FUNCTION_BLOCK CounterSp (* Basic Function Block Type *)
  (* Standard: 61499-2 *)
  (* Version 0.0, 7/15/2026, Schneider Electric, Template *)
  PACKAGE SE.Nereda;
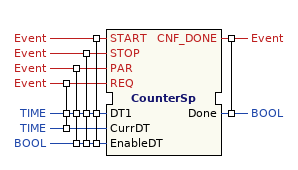
  EVENT_INPUT
    START WITH DT1, EnableDT; (* Normal Execution Request *)
    STOP WITH DT1, EnableDT;
    PAR WITH DT1, EnableDT;
    REQ WITH CurrDT, DT1;
  END_EVENT
  EVENT_OUTPUT
    CNF_DONE WITH Done; (* Execution Confirmation *)
  END_EVENT
  VAR_INPUT
    DT1 : TIME; (* Input event qualifier *)
    CurrDT : TIME;
    EnableDT : BOOL;
  END_VAR
  VAR_OUTPUT
    Done : BOOL; (* Output event qualifier *)
  END_VAR
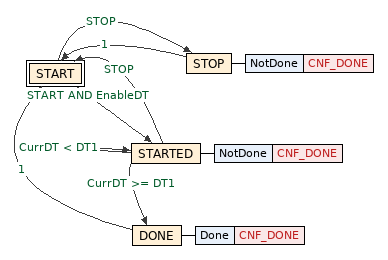
  EC_STATES
    START; (* Initial State *)
    STARTED : NotDone -> CNF_DONE; (* Normal execution *)
    DONE : Done -> CNF_DONE;
    STOP : NotDone -> CNF_DONE;
  END_STATES
  EC_TRANSITIONS
    START TO STARTED := START AND EnableDT;
    STARTED TO STARTED := CurrDT < DT1;
    STARTED TO DONE := CurrDT >= DT1;
    DONE TO START := 1;
    STARTED TO START := STOP;
    START TO STOP := STOP;
    STOP TO START := 1;
  END_TRANSITIONS
  ALGORITHM NotDone IN ST:
;
Done := FALSE;
  END_ALGORITHM
  ALGORITHM Done IN ST:
;
Done := TRUE;
  END_ALGORITHM
END_FUNCTION_BLOCK
